// TwinCAT 3 PLC project Plc1
// ProgramVersion: 3.1.4022.2
// libraries:
//   log4TC, * (mbc engineering GmbH)
//   Tc2_Standard, * (Beckhoff Automation GmbH)
//   Tc2_System, * (Beckhoff Automation GmbH)
//   Tc2_Utilities, * (Beckhoff Automation GmbH)
//   Tc3_Module, * (Beckhoff Automation GmbH)
// project tree:
//   / FB_LogTaskCycleTime.TcPOU (not stored), MAIN.TcPOU, PlcTask.TcTTO (not stored), PRG_SimulatedControlPlant.TcPOU, PRG_SimulateLoad.TcPOU, PRG_SimulateLogs.TcPOU
//   Utils/ FB_Plant.TcPOU, FB_PT1.TcPOU

// ---- MAIN.TcPOU
PROGRAM MAIN
VAR
	fbCycleTimeLogger	: FB_LogTaskCycleTime := (nCycleInterval:=1000);
END_VAR

IF _TaskInfo[1].FirstCycle THEN
	// Change AMS id if log service runs on different server than
	// plc. Remove if plc and service runs on the same machine.
	//PRG_TaskLog.Init('192.168.56.1.1.1');
	F_Log(E_LogLevel.eInfo, 'Plc started.');
END_IF

// simulates load on the task
PRG_SimulateLoad();

// simulate logs
PRG_SimulateLogs();

// logs the cycle time statistics
fbCycleTimeLogger();

// Simulates a PI controlled plant
PRG_SimulatedControlPlant();

PRG_TaskLog.Call();

END_PROGRAM

// ---- PRG_SimulateLoad.TcPOU
PROGRAM PRG_SimulateLoad
VAR
	nIdx	: UDINT;
	fResult	: REAL;
	fbRand	: DRAND := (Seed:=42);
	fRandom	: LREAL;
END_VAR

fbRand(Num=>fRandom);

FOR nIdx := 0 TO LREAL_TO_UDINT(fRandom * 10000) + 10000 DO
	fResult := SIN(UDINT_TO_REAL(nIdx));
END_FOR

END_PROGRAM

// ---- PRG_SimulateLogs.TcPOU
PROGRAM PRG_SimulateLogs
VAR
	fbRand	: DRAND := (Seed:=4242);
	nError	: INT;
END_VAR

fbRand();

IF fbRand.Num > 0.95 THEN
	IF fbRand.Num > 0.99 THEN
		nError := LREAL_TO_INT((1 - fbRand.Num) * 10000);
		F_LogLA1(E_LogLevel.eWarn, 'PRG_SimulatedLogs', 'Something bad happens. ErrorCode={code}', nError);
	ELSE
		F_LogL(E_LogLevel.eInfo, 'PRG_SimulatedLogs', 'Execution succeeded.');
	END_IF
END_IF

END_PROGRAM

// ---- PRG_SimulatedControlPlant.TcPOU
(* Simulation eines PI-Reglers mit Regelstrecke. *)
PROGRAM PRG_SimulatedControlPlant
VAR CONSTANT
	fInRangeWindow		: REAL := 0.1;
END_VAR
VAR
	fbPlant				: FB_Plant;
	fbController		: Tc2_Utilities.FB_BasicPID := (fKp:=0.7, fTn:=50, fTv:=0, fTd:=1E38);
	nLastControlError	: UINT;	
	bInRange			: BOOL;
	fbLogInterval		: TON := (PT:=T#1s);
END_VAR

IF _TaskInfo[1].FirstCycle THEN	
	// simualte a new setpoint value
	fbController.fSetpointValue := 10;
END_IF

// PI-Control
fbController(
	fActualValue	:= fbPlant.fActualOutput,
	fCtrlCycleTime  := 0.1,
);

// Logs the error code of the FB_BasicPID
IF fbController.nErrorStatus <> nLastControlError THEN
	nLastControlError := fbController.nErrorStatus;
	
	IF fbController.nErrorStatus > 0 THEN
		F_LogLA1(
			E_LogLevel.eError,
			'PRG_SimulatedControlPlant',
			'Error calling Basic-PID controller. Error={nErrorStatus}',
			fbController.nErrorStatus
		);
	END_IF
END_IF

// logs if the actual value is outside/inside of the setpoint
IF bInRange THEN
	IF ABS(fbController.fSetpointValue - fbController.fActualValue) > fInRangeWindow THEN
		F_LogLA1(
			E_LogLevel.eWarn,
			'PRG_SimulatedControlPlant',
			'Actual value is out of range ({setpoint}).',
			fbController.fSetpointValue
		);
		bInRange := FALSE;
	END_IF
ELSE
	IF ABS(fbController.fSetpointValue - fbController.fActualValue) <= fInRangeWindow THEN
		F_LogLA1(
			E_LogLevel.eInfo,
			'PRG_SimulatedControlPlant',
			'Actual value is in range of setpoint ({setpoint}).',
			fbController.fSetpointValue
		);
		bInRange := TRUE;
	END_IF
END_IF

// logs setpoint/actual value
fbLogInterval(IN:=NOT fbLogInterval.Q);
IF fbLogInterval.Q THEN
	F_LogLA2(
		E_LogLevel.eDebug, 
		'PRG_SimulatedControlPlant.Values', 
		'Setpoint={setpoint} Actual Value={actualvalue}',
		fbController.fSetpointValue,
		fbController.fActualValue
	);
END_IF
	
// Plant (simulated)
fbPlant(
	fControlInput	:= fbController.fCtrlOutput,
);

END_PROGRAM

// ---- Utils/FB_Plant.TcPOU
FUNCTION_BLOCK FB_Plant
VAR_INPUT
	fControlInput		: REAL;
END_VAR
VAR_OUTPUT
	fActualOutput		: REAL;
END_VAR
VAR
	fbPart1				: FB_PT1 := (fT1 := T#3S);
	fbPart2				: FB_PT1 := (fP := 2.4, fT1 := T#10s);				
END_VAR


fbPart1(
	fInput := fControlInput
);

fbPart2(
	fInput := fbPart1.fOutput
);

fActualOutput := fbPart2.fOutput;

END_FUNCTION_BLOCK

// ---- Utils/FB_PT1.TcPOU
FUNCTION_BLOCK FB_PT1
VAR_INPUT
	fInput		: REAL;
	fP			: REAL := 1.0;
	fT1			: TIME;
END_VAR
VAR_OUTPUT
	fOutput		: REAL;
END_VAR
VAR
	bInit		: BOOL;
END_VAR

IF NOT bInit THEN
	bInit := TRUE;
	fOutput := fInput;
END_IF

fOutput := fOutput + fP * (fInput - fOutput) * (1 / (TIME_TO_REAL(fT1) * 1E4 / UDINT_TO_REAL(_TaskInfo[Tc2_Utilities.GETCURTASKINDEXEX()].CycleTime) + 1));

END_FUNCTION_BLOCK
